FUNCTION_BLOCK FIELDBUS_WORD_TO_SIGNAL (* Mirrors IN->OUT if Signal Valid. *)
  (* Standard: 61499-1; Description: Copyright (c) 2026 HR Agrartechnik GmbH This program and the accompanying materials are made available under the terms of the Eclipse Public License 2.0 which is available at https://www.eclipse.org/legal/epl-2.0/ SPDX-License-Identifier: EPL-2.0 *)
  (* Version 1.0, 2026-05-30, Franz Höpfinger, HR Agrartechnik GmbH *)
  PACKAGE logiBUS::signalprocessing::fieldbus;
  IMPORT signalprocessing::FIELDBUS_SIGNAL::NOT_AVAILABLE_WM;
  IMPORT signalprocessing::FIELDBUS_SIGNAL::VALID_SIGNAL_W;
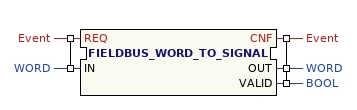
  EVENT_INPUT
    REQ WITH IN; (* Normal Execution Request *)
  END_EVENT
  EVENT_OUTPUT
    CNF WITH OUT, VALID; (* Execution Confirmation *)
  END_EVENT
  VAR_INPUT
    IN : WORD := NOT_AVAILABLE_WM; (* Input *)
  END_VAR
  VAR_OUTPUT
    OUT : WORD := 16#0000; (* Output Filtered *)
    VALID : BOOL := FALSE; (* TRUE if Signal is VALID *)
  END_VAR
  EC_STATES
    REQ : REQ -> CNF;
  END_STATES
  ALGORITHM REQ IN ST: (* Executed algorithm *)
IF (WORD_TO_UINT(IN) <= WORD_TO_UINT(VALID_SIGNAL_W)) THEN
	OUT := IN;
	VALID := BOOL#TRUE;
ELSE
	OUT := WORD#0;
	VALID := BOOL#FALSE;
END_IF;
  END_ALGORITHM
END_FUNCTION_BLOCK
